(*
	Add command by order, queue will scan only the head, this can be changed in the future.
	Element type type should be with a struct which contains DelayInfo_typ at start.  
*)

FUNCTION_BLOCK FB_CmdQueue
VAR_INPUT
	
	pBufferPool		: PVOID;
	BufferSize		: UDINT;
	ElementSize		: UDINT;
	rLogMsg 		: REFERENCE TO LogMsg ;
	Name : STRING := 'CmdQueue';			
	Position	:ULINT;
END_VAR
VAR_OUTPUT
END_VAR
VAR

	InitDone : BOOL;
	NumElements : UDINT;
	
	HeadIndex : UDINT; // index from 0
	TailIndex : UDINT; // index from 0
	UsedSize  : UDINT;
		
	MutexFlag : BOOL;
	
END_VAR

VAR_STAT
END_VAR

IF NOT InitDone THEN
	mInit();
	InitDone := TRUE;
END_IF

METHOD PUBLIC mAdd : BOOL
VAR_INPUT
	pElement		: PVOID;
END_VAR

VAR
	NewElementIndex : UDINT;
	
	pDelayedCmdInfo : POINTER TO DelayInfo_typ;
END_VAR

VAR_STAT
    sRid : UDINT := 1111;
END_VAR

IF NOT TestAndSet(MutexFlag) THEN
	RETURN;
END_IF

IF mIsFull() THEN
	MutexFlag := FALSE;
	RETURN;
END_IF

IF mIsEmpty() THEN
	NewElementIndex := TailIndex;	
ELSE
	NewElementIndex := (TailIndex + 1) MOD NumElements;
END_IF

TailIndex := NewElementIndex;
UsedSize := UsedSize + 1;

pDelayedCmdInfo := pElement;
pDelayedCmdInfo^.GroupId := pDelayedCmdInfo^.RequestId := sRid;
sRid := sRid+1;

IF (pDelayedCmdInfo^.pExecuted <> 0) THEN
//	pDelayedCmdInfo^.pExecuted^ := FALSE;
END_IF

pDelayedCmdInfo^.Executed := FALSE;
pDelayedCmdInfo^.LagError := 0;

MEMCPY((pBufferPool + NewElementIndex * ElementSize), pElement, ElementSize);

MutexFlag := FALSE;

mAdd := TRUE;
END_METHOD

METHOD PUBLIC mCheck : PVOID // will return true only when next cmd will be ready (time/pos is up)
VAR_INPUT
END_VAR

IF NOT TestAndSet(MutexFlag) THEN
	RETURN;
END_IF

IF mIsEmpty() THEN
	MutexFlag := FALSE;
	RETURN;
END_IF

IF NOT mCheckHead() THEN
	MutexFlag := FALSE;
	RETURN;
END_IF


mCheck := pBufferPool + HeadIndex * ElementSize;

UsedSize := UsedSize - 1;
IF NOT mIsEmpty() THEN
	HeadIndex := (HeadIndex + 1) MOD NumElements;	
END_IF



MutexFlag := FALSE;
END_METHOD

METHOD PRIVATE mCheckHead : BOOL
VAR_INPUT
END_VAR
VAR
	pDelayedCmdInfo : POINTER TO DelayInfo_typ;
	LogStr : STRING;
END_VAR
VAR_INST
	CmdTimer : StopWatch;
END_VAR

IF mIsEmpty() THEN
	RETURN;
END_IF

pDelayedCmdInfo := (pBufferPool + (HeadIndex * ElementSize));


CASE pDelayedCmdInfo^.DelayType OF
			
	eDelayType.Immediate: 
		mCheckHead := TRUE;
	
	eDelayType.DelayByPos:
		
		IF (Position >= pDelayedCmdInfo^.DelayValue) THEN
			LogStr := CONCAT(Name, 'rid=');
			LogStr := CONCAT(LogStr , UDINT_TO_STRING(pDelayedCmdInfo^.RequestId));
			LogStr := CONCAT(LogStr , ', now=');
			LogStr := CONCAT(LogStr , ULINT_TO_STRING(Position));
			LogStr := CONCAT(LogStr , ', target=');
			LogStr := CONCAT(LogStr , ULINT_TO_STRING(pDelayedCmdInfo^.DelayValue));
			fnLogMsg(ADR(rLogMsg), LOG_INFO, LogStr,0,0,0);
			pDelayedCmdInfo^.LagError := ULINT_TO_UDINT(Position - pDelayedCmdInfo^.DelayValue);
			mCheckHead := TRUE;
		END_IF
		
	eDelayType.DelayByTimer: 
	
		IF NOT CmdTimer.IsActive() THEN
			CmdTimer.Start();
		END_IF
		
		IF TIME_TO_ULINT(CmdTimer.ElapledTime()) >= pDelayedCmdInfo^.DelayValue THEN
			mCheckHead := TRUE;
		END_IF
	
END_CASE

IF mCheckHead THEN
	pDelayedCmdInfo^.Executed := TRUE;
	IF (pDelayedCmdInfo^.pExecuted <> 0) THEN
		pDelayedCmdInfo^.pExecuted^ := TRUE;
	END_IF
	
	IF pDelayedCmdInfo^.DelayType <> eDelayType.DelayByTimer THEN
		CmdTimer.Stop();
	END_IF

END_IF
END_METHOD

METHOD PUBLIC mClear : BOOL
VAR_INPUT
END_VAR
IF NOT TestAndSet(MutexFlag) THEN
	RETURN;
END_IF

TailIndex := HeadIndex := 0;
UsedSize := 0;

mClear := TRUE;

MutexFlag := FALSE;
END_METHOD

METHOD PUBLIC mFront : PVOID // will return true only when next cmd will be ready (time/pos is up)
VAR_INPUT
END_VAR

IF NOT TestAndSet(MutexFlag) THEN
	RETURN;
END_IF

IF mIsEmpty() THEN
	MutexFlag := FALSE;
	RETURN;
END_IF

mFront := pBufferPool + HeadIndex * ElementSize;

MutexFlag := FALSE;
END_METHOD

METHOD PRIVATE mInit : BOOL
VAR_INPUT
END_VAR

mClear();

NumElements := BufferSize/ElementSize;

mInit := TRUE;
END_METHOD

METHOD PUBLIC mIsEmpty : BOOL
VAR_INPUT
END_VAR
mIsEmpty := (UsedSize = 0);
END_METHOD

METHOD PUBLIC mIsFull : BOOL
VAR_INPUT
END_VAR
mIsFull := (UsedSize >= NumElements);
END_METHOD

END_FUNCTION_BLOCK

(* stored: Version 1.1.0.1, ProductVersion 3.1.4024.3
   POU FB_CmdQueue: Id {801951d8-2c3b-091d-0922-37305643ba25}, SpecialFunc None
   Folder Private: Id {19b77cf7-7b5f-4407-9bd1-dca703491f98}
   Method mAdd: Id {8ca9d29a-d1d9-0829-1dfc-c7deb2c0d0e0}
   Method mCheck: Id {654bd1c8-5c49-0bf7-3c5f-b3d473e2cdcd}
   Method mCheckHead: Id {837a474c-a37b-0dd5-0cb7-c12946045866}
   Method mClear: Id {861d8040-955e-0d50-1662-d361a0515d7a}
   Method mFront: Id {2c51ce45-73b6-42af-95d7-190a32b05a50}
   Method mInit: Id {f22b009f-5a76-05bd-3965-f47946690ddc}
   Method mIsEmpty: Id {a0cf7736-9050-081a-036f-2210006d0b7f}
   Method mIsFull: Id {d81af924-5005-019b-3e1a-0893d1142726} *)
